PROGRAM myHMIPLCRECIPE
VAR
	cyc : st_manual;
	bCTest1 : BOOL;
END_VAR

IF cyc.cyl1 = 1 THEN
	bCTest1 := TRUE;
	ELSE bCTest1 := FALSE;
END_IF

END_PROGRAM

(* stored: Version 1.1.0.1, ProductVersion 3.1.4024.11
   POU myHMIPLCRECIPE: Id {a878a368-56fe-42e8-81de-5612b07feebd}, SpecialFunc None *)
